METHOD SetPosition : BOOL
VAR_INPUT
	rPosition : LREAL;
END_VAR
// Start request once
IF NOT bSetPosRequested THEN
    bSetPosExecute   := TRUE;   // rising edge
    bSetPosRequested := TRUE;
END_IF

fbSetPos(Axis := Axis, Execute := bSetPosExecute, Position := rPosition, Mode := FALSE);

// Drop execute after it was accepted
IF fbSetPos.Busy THEN
    bSetPosExecute := FALSE;
END_IF

// Error handling
IF fbSetPos.Error THEN
    bSetPosExecute   := FALSE;
    bSetPosRequested := FALSE;   // ou mantenha TRUE se quiser retry controlado
    stStatus.eState  := E_ActuatorState.eError;
    stStatus.sMessage := 'Error in motor Set Position';
    SetPosition := FALSE;
    RETURN;
END_IF

// SUCCESS only on Done
IF fbSetPos.Done THEN
    bSetPosExecute   := FALSE;
    bSetPosRequested := FALSE;
    SetPosition := TRUE;
ELSE
    SetPosition := FALSE;
END_IF

(* Before Feb05th 2026
// Reuse the same logic from MoveAbsolute
IF NOT bSetPosRequested THEN
    bSetPosExecute := TRUE;
    bSetPosRequested := TRUE;
END_IF

// Call the internal motion block
fbSetPos(Axis := Axis, Execute := bSetPosExecute, Position := rPosition, Mode := FALSE);

// Update actuator status
stStatus.bBusy := fbSetPos.Busy;
stStatus.bDone := fbSetPos.Done;
stStatus.bError := fbSetPos.Error;
stStatus.iErrorCode := fbSetPos.ErrorID;

IF fbSetPos.busy THEN
    bSetPosExecute := FALSE;
END_IF

IF fbSetPos.Error THEN
    stStatus.eState := E_ActuatorState.eError;
    stStatus.sMessage := 'Error in motor Set Position';
END_IF

IF bSetPosRequested AND NOT fbSetPos.Busy AND NOT fbSetPos.Error THEN
    bSetPosRequested := FALSE;
    SetPosition := TRUE;
    RETURN;
ELSE
    SetPosition := FALSE;
END_IF
(*
// Call the internal motion block
fbSetPos(Axis := Axis, Execute := bSetPosExecute, Position := rPosition, Mode := FALSE);
*)*)
END_METHOD

METHOD Stop : BOOL
VAR_INPUT
END_VAR
VAR
END_VAR
// Default output value
Stop := FALSE;

// ============================================================================
// 1) First Stop trigger: set the request flag and generate the rising edge
//    on Execute for MC_Stop
// ============================================================================
IF NOT bStopRequested THEN
    bStopExecute  := TRUE;   // rising edge on MC_Stop.Execute
    bStopRequested := TRUE;
    bStopDone     := FALSE;
END_IF

// ============================================================================
// 2) Safety-net: if Stop was requested but the MC_Stop FB is idle,
//    without Done/Error, and Execute is FALSE (e.g., after a Reset),
//    then re-arm Execute to avoid getting stuck.
// ============================================================================
IF bStopRequested
   AND NOT fbStop.Busy
   AND NOT fbStop.Done
   AND NOT fbStop.Error
   AND NOT bStopExecute THEN
    bStopExecute := TRUE;
END_IF

// ============================================================================
// 3) Call the MC_Stop function block
// ============================================================================
fbStop(Axis := Axis, Execute := bStopExecute);

// ============================================================================
// 4) Internal Stop completion logic (Done / Requested)
// ============================================================================
IF fbStop.Done THEN
    bStopExecute := FALSE;      // release Execute after Done
    bStopDone    := TRUE;
END_IF

IF bStopDone AND NOT fbStop.Busy THEN
    bStopRequested := FALSE;    // stop procedure fully completed
END_IF

// ============================================================================
// 5) Error handling
// ============================================================================
stStatus.bError     := fbStop.Error;
stStatus.iErrorCode := fbStop.ErrorID;

IF fbStop.Error THEN
    stStatus.eState   := E_ActuatorState.eError;
    stStatus.sMessage := 'Error in Stop';
    // Stop remains FALSE; caller must handle Reset() afterwards
    RETURN;
END_IF

// ============================================================================
// 6) Successful completion: update status and return TRUE once
// ============================================================================
IF bStopDone AND NOT fbStop.Busy AND NOT bStopRequested THEN
    stStatus.bError     := FALSE;
    stStatus.iErrorCode := 0;
    stStatus.eState     := E_ActuatorState.eIdle;
    stStatus.sMessage   := 'Axis Stopped';

    // Prepare flags for the next Stop command
    bStopDone := FALSE;

    Stop := TRUE;   // Return TRUE for one cycle
    RETURN;
END_IF

// If execution reaches here, the Stop process is still ongoing
Stop := FALSE;


// Before - changed on Nov 20 2025
(* 
IF NOT bStopRequested THEN
	bStopExecute := TRUE;
	bStopRequested := TRUE;
END_IF

IF bStopRequested THEN
	fbStop(Axis := Axis, Execute := bStopExecute);
END_IF

IF bStopDone AND NOT fbStop.Busy THEN
	bStopRequested := FALSE;
END_IF

IF fbStop.Done THEN
	bStopExecute := FALSE;
	bStopDone := TRUE;
END_IF

stStatus.bError := fbStop.Error;
stStatus.iErrorCode := fbStop.ErrorID;

IF fbStop.Error THEN
	stStatus.eState := E_ActuatorState.eError;
	stStatus.sMessage := 'Error in Stop';
	Stop := FALSE;
END_IF

IF bStopDone AND NOT fbStop.Busy AND NOT bStopRequested THEN
	stStatus.bError := FALSE;
	stStatus.iErrorCode := 0;
	stStatus.eState := E_ActuatorState.eIdle;
	stStatus.sMessage := 'Axis Stopped';
	bStopDone := FALSE;
	Stop := TRUE;
	RETURN;
ELSE
	Stop := FALSE;
END_IF
*)
END_METHOD

END_FUNCTION_BLOCK

// ---- POUs/2. AutoCycle/Stages/FB_PostRun.TcPOU
FUNCTION_BLOCK FB_PostRun
VAR_INPUT
END_VAR
VAR_OUTPUT
END_VAR
VAR
END_VAR

END_FUNCTION_BLOCK

// ---- POUs/3. HMI/PRG_SetModulestatus.TcPOU
PROGRAM PRG_SetModulestatus
VAR
END_VAR

// Sets the Module status string based on the nTerminalState variable

// Terminal EK1100 EtherCAT Coupler
IF GVL_IO.nEK1100State = 8 THEN
	GVL_IO.sEK1100Status := 'Operational';
	ELSIF GVL_IO.nEK1100State = 4 THEN
 	GVL_IO.sEK1100Status := 'SAFEOP';
	ELSIF GVL_IO.nEK1100State = 3 THEN
 	GVL_IO.sEK1100Status := 'BOOT';
	ELSIF GVL_IO.nEK1100State = 2 THEN
 	GVL_IO.sEK1100Status := 'PREOP';
	ELSIF GVL_IO.nEK1100State = 1 THEN
 	GVL_IO.sEK1100Status := 'INIT';
END_IF

// TERMINAL - EL6070-0033	License Key Terminal for TwinCAT 3.1
IF GVL_IO.nEL6070State = 8 THEN
	GVL_IO.sEL6070Status := 'Operational';
	ELSIF GVL_IO.nEL6070State = 4 THEN
 	GVL_IO.sEL6070Status := 'SAFEOP';
	ELSIF GVL_IO.nEL6070State = 3 THEN
 	GVL_IO.sEL6070Status := 'BOOT';
	ELSIF GVL_IO.nEL6070State = 2 THEN
 	GVL_IO.sEL6070Status := 'PREOP';
	ELSIF GVL_IO.nEL6070State = 1 THEN
 	GVL_IO.sEL6070Status := 'INIT';
END_IF

// TERMINAL - EL6910 Safety PLC, 	Virtual Channels
IF GVL_IO.nEL6910State = 8 THEN
	GVL_IO.sEL6910Status := 'Operational';
	ELSIF GVL_IO.nEL6910State = 4 THEN
 	GVL_IO.sEL6910Status := 'SAFEOP';
	ELSIF GVL_IO.nEL6910State = 3 THEN
 	GVL_IO.sEL6910Status := 'BOOT';
	ELSIF GVL_IO.nEL6910State = 2 THEN
 	GVL_IO.sEL6910Status := 'PREOP';
	ELSIF GVL_IO.nEL6910State = 1 THEN
 	GVL_IO.sEL6910Status := 'INIT';
END_IF

// TERMINAL - EL1918_1 8-Channel Digital Safety Inputs
IF GVL_IO.nEL1918_1State = 8 THEN
	GVL_IO.sEL1918Status := 'Operational';
	ELSIF GVL_IO.nEL1918_1State = 4 THEN
 	GVL_IO.sEL1918Status := 'SAFEOP';
	ELSIF GVL_IO.nEL1918_1State = 3 THEN
 	GVL_IO.sEL1918Status := 'BOOT';
	ELSIF GVL_IO.nEL1918_1State = 2 THEN
 	GVL_IO.sEL1918Status := 'PREOP';
	ELSIF GVL_IO.nEL1918_1State = 1 THEN
 	GVL_IO.sEL1918Status := 'INIT';
END_IF

// TERMINAL - EL1918_2 8-Channel Digital Safety Inputs
IF GVL_IO.nEL1918_2State = 8 THEN
	GVL_IO.sEL1918_2Status := 'Operational';
	ELSIF GVL_IO.nEL1918_2State = 4 THEN
 	GVL_IO.sEL1918_2Status := 'SAFEOP';
	ELSIF GVL_IO.nEL1918_2State = 3 THEN
 	GVL_IO.sEL1918_2Status := 'BOOT';
	ELSIF GVL_IO.nEL1918_2State = 2 THEN
 	GVL_IO.sEL1918_2Status := 'PREOP';
	ELSIF GVL_IO.nEL1918_2State = 1 THEN
 	GVL_IO.sEL1918_2Status := 'INIT';
END_IF

// TERMINAL - EL2904 4-Channel Digital Output Terminal, TwinSAFE
IF GVL_IO.nEL2904State = 8 THEN
	GVL_IO.sEL2904Status := 'Operational';
	ELSIF GVL_IO.nEL2904State = 4 THEN
 	GVL_IO.sEL2904Status := 'SAFEOP';
	ELSIF GVL_IO.nEL2904State = 3 THEN
 	GVL_IO.sEL2904Status := 'BOOT';
	ELSIF GVL_IO.nEL2904State = 2 THEN
 	GVL_IO.sEL2904Status := 'PREOP';
	ELSIF GVL_IO.nEL2904State = 1 THEN
 	GVL_IO.sEL2904Status := 'INIT';
END_IF

// TERMINAL - EL2904_2 4-Channel Digital Output Terminal, TwinSAFE
IF GVL_IO.nEL2904_2State = 8 THEN
	GVL_IO.sEL2904_2Status := 'Operational';
	ELSIF GVL_IO.nEL2904_2State = 4 THEN
 	GVL_IO.sEL2904_2Status := 'SAFEOP';
	ELSIF GVL_IO.nEL2904_2State = 3 THEN
 	GVL_IO.sEL2904_2Status := 'BOOT';
	ELSIF GVL_IO.nEL2904_2State = 2 THEN
 	GVL_IO.sEL2904_2Status := 'PREOP';
	ELSIF GVL_IO.nEL2904_2State = 1 THEN
 	GVL_IO.sEL2904_2Status := 'INIT';
END_IF

// TERMINAL - EL1809_1 16-Channel Digital Input Terminal
IF GVL_IO.nEL1809State = 8 THEN
	GVL_IO.sEL1809Status := 'Operational';
	ELSIF GVL_IO.nEL1809State = 4 THEN
 	GVL_IO.sEL1809Status := 'SAFEOP';
	ELSIF GVL_IO.nEL1809State = 3 THEN
 	GVL_IO.sEL1809Status := 'BOOT';
	ELSIF GVL_IO.nEL1809State = 2 THEN
 	GVL_IO.sEL1809Status := 'PREOP';
	ELSIF GVL_IO.nEL1809State = 1 THEN
 	GVL_IO.sEL1809Status := 'INIT';
END_IF

// TERMINAL - EL2809_1	16-Channel Digital Output Terminal
IF GVL_IO.nEL2809State = 8 THEN
	GVL_IO.sEL2809Status := 'Operational';
	ELSIF GVL_IO.nEL2809State = 4 THEN
 	GVL_IO.sEL2809Status := 'SAFEOP';
	ELSIF GVL_IO.nEL2809State = 3 THEN
 	GVL_IO.sEL2809Status := 'BOOT';
	ELSIF GVL_IO.nEL2809State = 2 THEN
 	GVL_IO.sEL2809Status := 'PREOP';
	ELSIF GVL_IO.nEL2809State = 1 THEN
 	GVL_IO.sEL2809Status := 'INIT';
END_IF

// TERMINAL - EL3058	8-Channel Analog Input Terminal 4…20mA 12 Bit
IF GVL_IO.nEL3058State = 8 THEN
	GVL_IO.sEL3058Status := 'Operational';
	ELSIF GVL_IO.nEL3058State = 4 THEN
 	GVL_IO.sEL3058Status := 'SAFEOP';
	ELSIF GVL_IO.nEL3058State = 3 THEN
 	GVL_IO.sEL3058Status := 'BOOT';
	ELSIF GVL_IO.nEL3058State = 2 THEN
 	GVL_IO.sEL3058Status := 'PREOP';
	ELSIF GVL_IO.nEL3058State = 1 THEN
 	GVL_IO.sEL3058Status := 'INIT';
END_IF

// Terminal EL3058 8-Channel Analog Input Terminal 4…20mA 12 Bit (Term 10)
IF GVL_IO.nEL3058State = 8 THEN
	GVL_IO.sEL3058Status := 'Operational';
	ELSIF GVL_IO.nEL3058State = 4 THEN
 	GVL_IO.sEL3058Status := 'SAFEOP';
	ELSIF GVL_IO.nEL3058State = 3 THEN
 	GVL_IO.sEL3058Status := 'BOOT';
	ELSIF GVL_IO.nEL3058State = 2 THEN
 	GVL_IO.sEL3058Status := 'PREOP';
	ELSIF GVL_IO.nEL3058State = 1 THEN
 	GVL_IO.sEL3058Status := 'INIT';
END_IF

// Terminal EL6002	2-channel Serial Interface RS232, D-sub Connection (Term 11)
IF GVL_IO.nEL6002State = 8 THEN
	GVL_IO.sEL6002Status := 'Operational';
	ELSIF GVL_IO.nEL6002State = 4 THEN
 	GVL_IO.sEL6002Status := 'SAFEOP';
	ELSIF GVL_IO.nEL6002State = 3 THEN
 	GVL_IO.sEL6002Status := 'BOOT';
	ELSIF GVL_IO.nEL6002State = 2 THEN
 	GVL_IO.sEL6002Status := 'PREOP';
	ELSIF GVL_IO.nEL6002State = 1 THEN
 	GVL_IO.sEL6002Status := 'INIT';
END_IF

END_PROGRAM

// ---- POUs/7. EventsAndAlarms/FB_AlarmHandler.TcPOU
FUNCTION_BLOCK FB_AlarmHandler EXTENDS FB_TcAlarm
VAR_INPUT
	evtEntry	: TcEventEntry;
	bEvt		: BOOL;
	bConfirm	: BOOL;
	sSystem		: STRING; // Adding Alarm system name
	sMessage	: STRING; // Alarm Message
END_VAR
VAR_OUTPUT
END_VAR
VAR
	bInit	: BOOL := TRUE;
	bMem	: BOOL;
END_VAR

IF bInit THEN
	SUPER^.CreateEx(evtEntry, TRUE, 0);
	bInit	:= FALSE;
END_IF

// To when the alarm is triggered for the first time
IF bEvt AND NOT bMem AND SUPER^.eConfirmationState <> TcEventConfirmationState.WaitForConfirmation THEN
	SUPER^.ipArguments.AddString(sSystem).AddString(sMessage); // Adiciona as strings ao alarme
	SUPER^.Raise(0);
END_IF

// To when the alarm is reset
IF bMem AND NOT bEvt THEN
	SUPER^.Clear(0, FALSE);
END_IF

// Alarm confirmation
IF bConfirm THEN
	SUPER^.Confirm(0);
END_IF

bMem := bEvt;

END_FUNCTION_BLOCK

// ---- POUs/7. EventsAndAlarms/FB_ErrorHandler.TcPOU
FUNCTION_BLOCK FB_ErrorHandler

VAR_INPUT
END_VAR

VAR_OUTPUT
	bErrorResolved : BOOL;
END_VAR

VAR
END_VAR

//bErrorResolved := (* Verdadeiro quando o erro for resolvido

END_FUNCTION_BLOCK

// ---- POUs/Functions/F_REAL_TO_STRING_2DEC.TcPOU
FUNCTION F_REAL_TO_STRING_2DEC : STRING
VAR_INPUT
	rInput : REAL;
END_VAR
VAR
	iInt    : DINT;
    iDec    : DINT;
    rTmp    : REAL;
END_VAR

iInt := TRUNC(rInput);
rTmp := ABS(rInput - iInt);            // decimal part
iDec := TRUNC((rTmp * 100.0) + 0.5);   // manual rounding

IF rInput >= 0.0 THEN
    F_REAL_TO_STRING_2DEC := CONCAT( DINT_TO_STRING(iInt), CONCAT('.', DINT_TO_STRING(iDec)) );
ELSE
    F_REAL_TO_STRING_2DEC := CONCAT('-', CONCAT( DINT_TO_STRING(ABS(iInt)), CONCAT('.', DINT_TO_STRING(iDec)) ));
END_IF

END_FUNCTION

// ---- POUs/Functions/F_SqlEscapeString.TcPOU
FUNCTION F_SqlEscapeString : STRING
VAR_INPUT
	sInput : STRING(500);
END_VAR
VAR
	i       : INT;
    sChar   : STRING(1);
    sOutput : STRING(500);
END_VAR

sOutput := '';

FOR i := 1 TO LEN(sInput) DO
    sChar := MID(sInput, 1, i);

    IF sChar = '$'' THEN
        sOutput := CONCAT(sOutput, '$'$'');
    ELSE
        sOutput := CONCAT(sOutput, sChar);
    END_IF
END_FOR

F_SqlEscapeString := sOutput;

END_FUNCTION

// ---- POUs/Levels/FB_LevelSensors.TcPOU
FUNCTION_BLOCK FB_LevelSensors
VAR_INPUT
	abyInputs : ARRAY[1..5, 0..3] OF BYTE; // 5 sensors, 4 bytes each
    eSensorID : E_LevelSensorID;
END_VAR
VAR_OUTPUT
	stLevelData : ST_KQ1000_Data;
END_VAR
VAR
	fbParsers : ARRAY[1..5] OF FB_KQ1000_Parser;
    i : INT;
END_VAR

// Parsers execute
FOR i := 1 TO 5 DO
    fbParsers[i].byInput0 := abyInputs[i, 0];
    fbParsers[i].byInput1 := abyInputs[i, 1];
    fbParsers[i].byInput2 := abyInputs[i, 2];
    fbParsers[i].byInput3 := abyInputs[i, 3];
END_FOR

// Sends the result based on sensor id
stLevelData := fbParsers[eSensorID].stData;

END_FUNCTION_BLOCK

// ---- POUs/MARCO/OLD/POU_Master_Calib.TcPOU
PROGRAM POU_Master_Calib
VAR
	criteria: REAL := 0.5; // Acceptance Criteria (0.1 ~ 5.0)
	failures: INT := 0; // Allowable Failures (0 ~ 5)
	targetVolume: REAL := 0.50; // Volume Target (mL)
	replicates: INT := 2; // Number of checks (0 ~ 10)
	tareWt: REAL; //Weight before
	grossWt: REAL; //Weight after
	netWt: REAL; // rsult of (grossWt - tareWt)
	netVolume: REAL; //result of (netWt * density)
	state: INT;
	valveNo: INT;
	pumpNo: INT:=1;
	timeWt: ton;
	timer2: ton;
	timer3: ton;
	selectPump: ARRAY[1..10] OF STRING;
	result: ARRAY[1..10] OF ST_Results;
	start: BOOL;
	stop: BOOL;
	movimentDONE: BOOL;
	revs: REAL;
	valvePos: USINT;
	repli: INT:= 1;
	axiPower: MC_Power;
	i: INT;
	scale: FB_ScaleDevice;
	adjust: ARRAY[1..10] OF BOOL;
	correctRev: REAL;
	enableAdj: BOOL;
	opening: REAL;
	runLinear: BOOL;
	adjustSum: REAL;
	recResult: int:=1;
END_VAR

timeWt();
timer2();
timer3();

IF stop THEN
	powerOFF();
	stop:=FALSE;
END_IF

IF pumpNo = 1 OR pumpNo = 2 THEN
	valveNo:= 1;
ELSIF pumpNo = 3 OR pumpNo = 4 THEN
	valveNo:= 2;
ELSIF pumpNo = 5 OR pumpNo = 6 THEN
	valveNo:= 3;
ELSIF pumpNo = 7 OR pumpNo = 8 THEN
	valveNo:= 4;
ELSIF pumpNo = 9 OR pumpNo = 10 THEN
	valveNo:= 5;
END_IF

CASE state OF
	
0: //Idle
	IF start THEN
		GVL_Marco.revs:= GVL_Marco.mL_target;
		GVL_Marco.valvPos:= 6;
		timeWt(in:=TRUE, pt:=T#10S);
		repli:= 1;
		recResult:= 1;
		
		FOR i:= 1 TO 10 BY 1 DO
			GVL_Marco.resetAxi[i]:= FALSE;
			GVL_Marco.enableAxi[i]:= TRUE;
		END_FOR 
		
		FOR i:= 1 TO 5 BY 1 DO
			GVL_Marco.enableValv[i]:= TRUE;		
		END_FOR
		
		FOR i:=1 TO 50 BY 1 DO
			GVL_Marco.calibResult[i].grossWt:=0;
			GVL_Marco.calibResult[i].netWt:=0;
			GVL_Marco.calibResult[i].pumpNo:=0;
			GVL_Marco.calibResult[i].tareWt:=0;
		END_FOR
		
		state:= 10;
	ELSE
		state:= 0;
	END_IF
	
10:	//Disable valves
	
	IF GVL_Motion.aValves[1].Axis.Status.InTargetPosition AND
		GVL_Motion.aValves[2].Axis.Status.InTargetPosition AND
		GVL_Motion.aValves[3].Axis.Status.InTargetPosition AND
		GVL_Motion.aValves[4].Axis.Status.InTargetPosition AND
		GVL_Motion.aValves[5].Axis.Status.InTargetPosition AND timeWt.Q THEN
		FOR i:= 1 TO 5 BY 1 DO
			GVL_Marco.enableValv[i]:= FALSE;		
		END_FOR
		timeWt(in:=FALSE);
		timer3(in:=TRUE, pt:=T#10S);
		state:= 20;
	ELSE
		state:= 10;
	END_IF		

20:	//Fill Jar from Box
	
	IF NOT GVL_Motion.aPumps[pumpNo].Rotary.Axis.Status.Disabled AND (timer3.Q OR timeWt.Q) THEN
		IF repli < 2 THEN
		revs:= GVL_Marco.revs*2.4;	
		END_IF
		GVL_Marco.runFWD[pumpNo]:= TRUE;
		timer3(in:=FALSE);
		start:= FALSE;
		timer2(in:=TRUE, pt:=T#10S);
		state:= 30;
	ELSE
		state:= 20;
	END_IF

30: //Waiting

	IF GVL_Motion.aPumps[pumpNo].Rotary.Axis.Status.NotMoving AND timer2.Q THEN
		GVL_Marco.runFWD[pumpNo]:= FALSE;
		timer2(in:=FALSE);
		timeWt(in:=TRUE, pt:=T#10S);
		GVL_Calibration.fbScaleDevice.RequestWeight();
		state:= 40;
	ELSE
		state:= 30;
	END_IF
	
40: //Make Tara
	
	IF timeWt.Q THEN
		tareWt:= GVL_Calibration.fbScaleDevice.RequestWeight();
		timeWt(in:=FALSE);
		state:= 50;
	ELSE
		state:= 40;
	END_IF
	
50: //Fill box from jar

	IF tareWt <> 9999.0 THEN
		GVL_Marco.calibResult[recResult].tareWt:= tareWt;
		revs:= GVL_Marco.revs;
		GVL_Marco.runBWD[pumpNo]:= TRUE;
		timer2(in:=TRUE, pt:=T#10S);
		state:= 60;
	ELSE
		state:= 50;
	END_IF
	
60: //Waiting

	IF NOT GVL_Motion.aPumps[pumpNo].Rotary.Axis.Status.Moving AND timer2.Q THEN
		GVL_Marco.runBWD[pumpNo]:= FALSE;
		timer2(in:=FALSE);
		timeWt(in:=TRUE, pt:=T#10S);
		GVL_Calibration.fbScaleDevice.RequestWeight();
		state:= 70;
	ELSE
		state:= 60;
	END_IF

70: //Get gross weight
	
	IF timeWt.Q THEN
		grossWt:= GVL_Calibration.fbScaleDevice.RequestWeight();
		timeWt(in:=FALSE);
		state:= 80;
	ELSE
		state:= 70;
	END_IF
	
80: //Return jar to box

	IF grossWt <> 9999.0 THEN
		GVL_Marco.calibResult[recResult].grossWt:= grossWt;
		GVL_Marco.calibResult[recResult].netWt:= GVL_Marco.calibResult[recResult].grossWt - GVL_Marco.calibResult[recResult].tareWt;
		GVL_Marco.calibResult[recResult].pumpNo:= pumpNo;
		recResult:= recResult +1;
			
		//revs:= GVL_Marco.revs;
		//GVL_Marco.runFWD[pumpNo]:= TRUE;

		timer3(in:=TRUE, pt:=T#10S);
		repli := repli +1; 
		state:= 90;
	ELSE
		state:= 80;
	END_IF

90: //Check replicates

	IF repli < replicates+1 AND timer3.Q AND GVL_Motion.aPumps[pumpNo].Rotary.Axis.Status.NotMoving THEN //Return to the next replicate
		timer3(in:=FALSE);
		timeWt(in:=TRUE, pt:=T#10S);
		GVL_Marco.runFWD[pumpNo]:= FALSE;
		state:= 20;
	ELSIF repli >= replicates AND timer3.Q AND GVL_Motion.aPumps[pumpNo].Rotary.Axis.Status.NotMoving THEN //Empty the jar to box
		timer3(in:=FALSE);
		GVL_Marco.runFWD[pumpNo]:= FALSE;
		revs:= GVL_Marco.revs*2.4;
		GVL_Marco.runBWD[pumpNo]:= TRUE;
		timer2(in:=TRUE, pt:=T#10S);
		state:= 100;
	ELSE
		state:= 90;
	END_IF

100: 

	IF  GVL_Motion.aPumps[pumpNo].Rotary.Axis.Status.NotMoving AND timer2.Q THEN
		timer2(in:=FALSE);
		IF pumpNo = 10 THEN
			GVL_Marco.runBWD[pumpNo]:= FALSE;
			timer3(in:=TRUE, pt:=T#10S);
			state:= 110;
		ELSE
			pumpNo:= pumpNo + 1;
			repli:= 1;
			timer3(in:=TRUE, pt:=T#10S);
			state:= 20;
		END_IF
		
	ELSE
		state:= 100;
	END_IF
	
110: //Done

	IF GVL_Motion.aPumps[1].Rotary.Axis.Status.NotMoving AND
		GVL_Motion.aPumps[2].Rotary.Axis.Status.NotMoving AND
		GVL_Motion.aPumps[3].Rotary.Axis.Status.NotMoving AND
		GVL_Motion.aPumps[4].Rotary.Axis.Status.NotMoving AND
		GVL_Motion.aPumps[5].Rotary.Axis.Status.NotMoving AND
		GVL_Motion.aPumps[6].Rotary.Axis.Status.NotMoving AND
		GVL_Motion.aPumps[7].Rotary.Axis.Status.NotMoving AND
		GVL_Motion.aPumps[8].Rotary.Axis.Status.NotMoving AND
		GVL_Motion.aPumps[9].Rotary.Axis.Status.NotMoving AND
		GVL_Motion.aPumps[10].Rotary.Axis.Status.NotMoving AND timer3.Q THEN
		FOR i:=1 TO 10 BY 1 DO
			GVL_Marco.runBWD[i]:= FALSE;
		END_FOR
		
		timer3(in:=FALSE);
		timeWt(in:=TRUE, pt:=T#10S);
		state:= 120;
	ELSE
		state:= 110;
	END_IF
	
120:

	IF GVL_Motion.aPumps[1].Rotary.Axis.Status.NotMoving AND
		GVL_Motion.aPumps[2].Rotary.Axis.Status.NotMoving AND
		GVL_Motion.aPumps[3].Rotary.Axis.Status.NotMoving AND
		GVL_Motion.aPumps[4].Rotary.Axis.Status.NotMoving AND
		GVL_Motion.aPumps[5].Rotary.Axis.Status.NotMoving AND
		GVL_Motion.aPumps[6].Rotary.Axis.Status.NotMoving AND
		GVL_Motion.aPumps[7].Rotary.Axis.Status.NotMoving AND
		GVL_Motion.aPumps[8].Rotary.Axis.Status.NotMoving AND
		GVL_Motion.aPumps[9].Rotary.Axis.Status.NotMoving AND
		GVL_Motion.aPumps[10].Rotary.Axis.Status.NotMoving AND timeWt.Q THEN
		FOR i:=1 TO 10 BY 1 DO
			GVL_Marco.resetAxi[i]:= TRUE;
			GVL_Marco.enableAxi[i]:= FALSE;
		END_FOR
		
		(*IF GVL_Marco.revs > GVL_Marco.mL_target THEN
			correctRev:= GVL_Marco.revs - GVL_Marco.mL_target;
		ELSIF GVL_Marco.revs < GVL_Marco.mL_target THEN
			correctRev:= GVL_Marco.mL_target - GVL_Marco.revs; 	
		END_IF*)
		state:= 0;
	ELSE
		state:= 120;
	END_IF
	
END_CASE

METHOD moveValve : BOOL
VAR
	state: INT;
	valveNo: INT;
END_VAR
VAR_INPUT
	pumNo: INT;
	valvePos: USINT;
	
END_VAR
IF pumpNo = 1 OR pumpNo = 2 THEN
	valveNo:= 1;
ELSIF pumpNo = 3 OR pumpNo = 4 THEN
	valveNo:= 2;
ELSIF pumpNo = 5 OR pumpNo = 6 THEN
	valveNo:= 3;
ELSIF pumpNo = 7 OR pumpNo = 8 THEN
	valveNo:= 4;
ELSIF pumpNo = 9 OR pumpNo = 10 THEN
	valveNo:= 5;
END_IF

GVL_Motion.aValvesObj[valveNo].MoveValve(iPosition := valvePos, rVelocity := GVL_Motion.aValves[1].rTargetVel, rAcc := GVL_Motion.aValves[1].rAcceleration, rDec := GVL_Motion.aValves[1].rDeceleration);

CASE state OF
	
0:

	IF NOT GVL_Motion.aValves[valveNo].Axis.Status.Moving THEN
		GVL_Motion.aValvesObj[valveNo].MoveValve(iPosition := valvePos, rVelocity := GVL_Motion.aValves[1].rTargetVel, rAcc := GVL_Motion.aValves[1].rAcceleration, rDec := GVL_Motion.aValves[1].rDeceleration);
		movimentDONE:=FALSE;
		state:= 1;
	ELSE
		state:= 0;	
	END_IF

1:
	IF NOT GVL_Motion.aValves[valveNo].Axis.Status.Moving THEN
			movimentDONE:= TRUE;
			State:= 0;
		ELSE
			state:= 1;
		END_IF
	
	
END_CASE
END_METHOD

METHOD powerOFF : BOOL
VAR
	axiPower: MC_Power;
	pumpNo: INT;
	
END_VAR
VAR_INPUT
	
	
END_VAR
FOR pumpNo:=1 TO 10 BY 1 DO
	axiPower(
	Axis:= GVL_Motion.aPumps[pumpNo].Rotary.Axis,
	Enable:= FALSE,
	Enable_Negative:= FALSE,
	Enable_Positive:= FALSE,
	Override:= 100);
	
	axiPower(
	Axis:= GVL_Motion.aPumps[pumpNo].Linear.Axis,
	Enable:= FALSE,
	Enable_Negative:= FALSE,
	Enable_Positive:= FALSE,
	Override:= 100);
END_FOR
END_METHOD

METHOD runBwd : BOOL
VAR
	moveRel: MC_MoveRelative;
	selectPosRel: LREAL;
	
END_VAR
VAR_INPUT
	pumpNo: INT;
	revs: INT;
	 
END_VAR

selectPosRel:= revs*360;

moveRel(
	Axis:= GVL_Motion.aPumps[pumpNo].Rotary.Axis,
	Execute:= TRUE,
	Distance:= selectPosRel*-1,
	Velocity:= 3000,
	Acceleration:= 3000,
	Deceleration:= 3000);
END_METHOD

METHOD runFwd : BOOL
VAR
	moveRel: MC_MoveRelative;
	selectPosRel: LREAL;
	
END_VAR
VAR_INPUT
	pumpNo: INT;
	revs: INT;
	 
END_VAR

selectPosRel:= revs*360;

moveRel(
	Axis:= GVL_Motion.aPumps[pumpNo].Rotary.Axis,
	Execute:= TRUE,
	Distance:= selectPosRel,
	Velocity:= 3000,
	Acceleration:= 3000,
	Deceleration:= 3000);
END_METHOD

END_PROGRAM

// ---- POUs/MARCO/OLD/POU_Master_Calib_1.TcPOU
PROGRAM POU_Master_Calib_1
VAR
	criteria: REAL := 0.5; // Acceptance Criteria (0.1 ~ 5.0)
	failures: INT := 0; // Allowable Failures (0 ~ 5)
	targetVolume: REAL := 0.50; // Volume Target (mL)
	replicates: INT := 5; // Number of checks (0 ~ 10)
	tareWt: REAL; //Weight before
	grossWt: REAL; //Weight after
	netWt: REAL; // rsult of (grossWt - tareWt)
	netVolume: REAL; //result of (netWt * density)
	state: INT;
	valveNo: INT;
	pumpNo: INT:=1;
	timeWt: ton;
	timer2: ton;
	timer3: ton;
	selectPump: ARRAY[1..10] OF STRING;
	result: ARRAY[1..50] OF ST_Results;
	start: BOOL;
	stop: BOOL;
	movimentDONE: BOOL;
	revs: REAL;
	valvePos: USINT;
	repli: INT:= 1;
	axiPower: MC_Power;
	i: INT;
	scale: FB_ScaleDevice;
	adjust: ARRAY[1..10] OF BOOL;
	correctRev: REAL;
	enableAdj: BOOL;
	opening: REAL;
	runLinear: BOOL;
	adjustSum: REAL;
END_VAR

timeWt();
timer2();
timer3();

IF stop THEN
	powerOFF();
	stop:=FALSE;
END_IF

IF pumpNo = 1 OR pumpNo = 2 THEN
	valveNo:= 1;
ELSIF pumpNo = 3 OR pumpNo = 4 THEN
	valveNo:= 2;
ELSIF pumpNo = 5 OR pumpNo = 6 THEN
	valveNo:= 3;
ELSIF pumpNo = 7 OR pumpNo = 8 THEN
	valveNo:= 4;
ELSIF pumpNo = 9 OR pumpNo = 10 THEN
	valveNo:= 5;
END_IF

CASE state OF
	
0: //Idle
	IF start THEN
		GVL_Marco.revs:= GVL_Marco.mL_target;
		GVL_Marco.resetAxi:= FALSE;
		GVL_Marco.valvPos:= 2;
		GVL_Marco.enableValv:= TRUE;
		timeWt(in:=TRUE, pt:=T#10S);
		GVL_Marco.enableAxi:= TRUE;
		FOR i:=1 TO 10 BY 1 DO
			result[i].gross:= 0;
			result[i].rest:= 0;
			result[i].tare:= 0;
		END_FOR
		repli:= 1;
		state:= 10;
	ELSE
		state:= 0;
	END_IF
	
10:	//Enable the pump motor
	
	IF GVL_Motion.aValves[valveNo].Axis.Status.InTargetPosition AND timeWt.Q THEN
		GVL_Marco.enableValv:= FALSE;
		timeWt(in:=FALSE);
		IF pumpNo >= 10 THEN
			pumpNo:= 2;
			state:= 20;
		ELSE
			pumpNo:= pumpNo + 1;
			state:= 0;
		END_IF
	ELSE
		state:= 10;
	END_IF		

20:	//Fill the Jars from Bottle
	
	IF NOT GVL_Motion.aPumps[pumpNo].Rotary.Axis.Status.Disabled AND timer2.Q THEN
		revs:= GVL_Marco.revs*2.4;
		GVL_Marco.runFWD:= TRUE;
		timer2(in:=TRUE, pt:=T#10S);
		IF pumpNo >= 10 THEN
			pumpNo:= 2;
			start:= FALSE;
			state:= 30;
		ELSE
			timer2(in:=FALSE);
			pumpNo:= pumpNo + 1;
			GVL_Marco.runFWD:= FALSE;
			state:= 20;
		END_IF
	ELSE
		state:= 20;
	END_IF

30: //Move valve to position 6
	
	IF NOT GVL_Motion.aPumps[pumpNo].Rotary.Axis.Status.Moving AND timer2.Q THEN
		GVL_Marco.runFWD:= FALSE;
		GVL_Marco.valvPos:= 6;
		GVL_Marco.enableValv:= TRUE;
		timer2(in:=FALSE);
		timeWt(in:=TRUE, pt:=T#10S);
		IF pumpNo >= 10 THEN
			pumpNo:= 2;
			state:= 40;
		ELSE
			pumpNo:= pumpNo + 1;
			state:= 30;
		END_IF
	ELSE
		state:= 30;
	END_IF


40: //Fill the calibration box( SETUP )

	IF GVL_Motion.aValves[valveNo].Axis.Status.InTargetPosition AND timeWt.Q THEN
		GVL_Marco.enableValv:= FALSE;
		revs:= GVL_Marco.revs/2;
		GVL_Marco.runBWD:= TRUE;
		timeWt(in:=FALSE);
		timer2(in:=TRUE, pt:=T#5S);
		state:= 50;
		
	ELSE
		state:= 40;	
	END_IF

50: //Waiting

	IF NOT GVL_Motion.aPumps[pumpNo].Rotary.Axis.Status.Moving AND timer2.Q THEN
		GVL_Marco.runBWD:= FALSE;
		timer2(in:=FALSE);
		timeWt(in:=TRUE, pt:=T#10S);
		GVL_Calibration.fbScaleDevice.RequestWeight();
		state:= 55;
	ELSE
		state:= 50;
	END_IF
	
55: //Make Tara
	
	IF timeWt.Q THEN
		tareWt:= GVL_Calibration.fbScaleDevice.RequestWeight();
		timeWt(in:=FALSE);
		state:= 60;
	ELSE
		state:= 55;
	END_IF
	
60: //Fill calibration box

	IF tareWt <> 9999.0 THEN
		result[repli].tare:= tareWt;
		revs:= GVL_Marco.revs;
		GVL_Marco.runBWD:= TRUE;
		timer2(in:=TRUE, pt:=T#5S);
		state:= 70;
	ELSE
		state:= 60;
	END_IF
	
70: //Waiting

	IF NOT GVL_Motion.aPumps[pumpNo].Rotary.Axis.Status.Moving AND timer2.Q THEN
		GVL_Marco.runBWD:= FALSE;
		timer2(in:=FALSE);
		timeWt(in:=TRUE, pt:=T#10S);
		GVL_Calibration.fbScaleDevice.RequestWeight();
		state:= 75;
	ELSE
		state:= 70;
	END_IF

75: //Get gross weight
	
	IF timeWt.Q THEN
		grossWt:= GVL_Calibration.fbScaleDevice.RequestWeight();
		timeWt(in:=FALSE);
		state:= 80;
	ELSE
		state:= 75;
	END_IF
	
80: //Return solvent to jar

	IF grossWt <> 9999.0 THEN
		result[repli].gross:= grossWt;
		result[repli].rest:= result[repli].gross - result[repli].tare;
		netWt:= result[repli].rest;
			IF (netWt > GVL_Marco.mL_target+((GVL_Marco.mL_target*0.5)/100) OR netWt < GVL_Marco.mL_target-((GVL_Marco.mL_target*0.5)/100)) THEN
				adjust[repli]:= TRUE;
			ELSE
				adjust[repli]:= FALSE;
			END_IF
			IF repli >= replicates THEN
				revs:= GVL_Marco.revs*2;
				GVL_Marco.runFWD:= TRUE;
			ELSE
				revs:= GVL_Marco.revs;
				GVL_Marco.runFWD:= TRUE;
			END_IF
		timer3(in:=TRUE, pt:=T#10S);
		repli := repli +1;
		state:= 90;
	ELSE
		state:= 80;
	END_IF

90: //Check replicates

	IF repli < replicates+1 AND timer3.Q AND GVL_Motion.aPumps[pumpNo].Rotary.Axis.Status.NotMoving THEN
		timer3(in:=FALSE);
		GVL_Marco.runFWD:= FALSE;
		timer2(in:=TRUE, pt:=T#5S);
		state:= 50;
	ELSIF repli >= replicates AND timer3.Q AND GVL_Motion.aPumps[pumpNo].Rotary.Axis.Status.NotMoving THEN
		timer3(in:=FALSE);
		GVL_Marco.runFWD:= FALSE;
		GVL_Marco.valvPos:= 2;
		GVL_Marco.enableValv:= TRUE;
		timer2(in:=TRUE, pt:=T#10S);
		IF pumpNo >= 10 THEN
			pumpNo:= 2;
			state:= 100;
		ELSE
			pumpNo:= pumpNo + 1;
			repli:= 1;
			state:= 50;
		END_IF
	ELSE
		state:= 90;
	END_IF

100: //Empty the jar

	IF  GVL_Motion.aValves[valveNo].Axis.Status.InTargetPosition AND timer2.Q THEN
		GVL_Marco.enableValv:= FALSE;
		revs:= GVL_Marco.revs*2.4;
		GVL_Marco.runBWD:= TRUE;
		timer2(in:=FALSE);
		timer3(in:=TRUE, pt:=T#10S);
		IF pumpNo >= 10 THEN
			pumpNo:= 2;
			state:= 110;
		ELSE
			pumpNo:= pumpNo + 1;
			state:= 100;
		END_IF
	ELSE
		state:= 100;
	END_IF
	
110: //Done

	IF NOT GVL_Motion.aPumps[pumpNo].Rotary.Axis.Status.Moving AND timer3.Q THEN
		GVL_Marco.runBWD:= FALSE;
		timer3(in:=FALSE);
		timeWt(in:=TRUE, pt:=T#10S);
		IF pumpNo >= 10 THEN
			pumpNo:= 2;
			state:= 120;
		ELSE
			pumpNo:= pumpNo + 1;
			state:= 110;
		END_IF
	ELSE
		state:= 110;
	END_IF
	
120:

	IF GVL_Motion.aPumps[pumpNo].Rotary.Axis.Status.NotMoving AND timeWt.Q THEN
		GVL_Marco.resetAxi:= TRUE;
		GVL_Marco.enableAxi:= FALSE;
		IF pumpNo >= 10 THEN
			pumpNo:= 2;
			state:= 0;
		ELSE
			pumpNo:= pumpNo + 1;
			state:= 120;
		END_IF
	ELSE
		state:= 120;
	END_IF
	
END_CASE

METHOD moveValve : BOOL
VAR
	state: INT;
	valveNo: INT;
END_VAR
VAR_INPUT
	pumNo: INT;
	valvePos: USINT;
	
END_VAR
IF pumpNo = 1 OR pumpNo = 2 THEN
	valveNo:= 1;
ELSIF pumpNo = 3 OR pumpNo = 4 THEN
	valveNo:= 2;
ELSIF pumpNo = 5 OR pumpNo = 6 THEN
	valveNo:= 3;
ELSIF pumpNo = 7 OR pumpNo = 8 THEN
	valveNo:= 4;
ELSIF pumpNo = 9 OR pumpNo = 10 THEN
	valveNo:= 5;
END_IF

GVL_Motion.aValvesObj[valveNo].MoveValve(iPosition := valvePos, rVelocity := GVL_Motion.aValves[1].rTargetVel, rAcc := GVL_Motion.aValves[1].rAcceleration, rDec := GVL_Motion.aValves[1].rDeceleration);

CASE state OF
	
0:

	IF NOT GVL_Motion.aValves[valveNo].Axis.Status.Moving THEN
		GVL_Motion.aValvesObj[valveNo].MoveValve(iPosition := valvePos, rVelocity := GVL_Motion.aValves[1].rTargetVel, rAcc := GVL_Motion.aValves[1].rAcceleration, rDec := GVL_Motion.aValves[1].rDeceleration);
		movimentDONE:=FALSE;
		state:= 1;
	ELSE
		state:= 0;	
	END_IF

1:
	IF NOT GVL_Motion.aValves[valveNo].Axis.Status.Moving THEN
			movimentDONE:= TRUE;
			State:= 0;
		ELSE
			state:= 1;
		END_IF
	
	
END_CASE
END_METHOD

METHOD powerOFF : BOOL
VAR
	axiPower: MC_Power;
	pumpNo: INT;
	
END_VAR
VAR_INPUT
	
	
END_VAR
FOR pumpNo:=1 TO 10 BY 1 DO
	axiPower(
	Axis:= GVL_Motion.aPumps[pumpNo].Rotary.Axis,
	Enable:= FALSE,
	Enable_Negative:= FALSE,
	Enable_Positive:= FALSE,
	Override:= 100);
	
	axiPower(
	Axis:= GVL_Motion.aPumps[pumpNo].Linear.Axis,
	Enable:= FALSE,
	Enable_Negative:= FALSE,
	Enable_Positive:= FALSE,
	Override:= 100);
END_FOR
END_METHOD

METHOD runBwd : BOOL
VAR
	moveRel: MC_MoveRelative;
	selectPosRel: LREAL;
	
END_VAR
VAR_INPUT
	pumpNo: INT;
	revs: INT;
	 
END_VAR

selectPosRel:= revs*360;

moveRel(
	Axis:= GVL_Motion.aPumps[pumpNo].Rotary.Axis,
	Execute:= TRUE,
	Distance:= selectPosRel*-1,
	Velocity:= 3000,
	Acceleration:= 3000,
	Deceleration:= 3000);
END_METHOD

METHOD runFwd : BOOL
VAR
	moveRel: MC_MoveRelative;
	selectPosRel: LREAL;
	
END_VAR
VAR_INPUT
	pumpNo: INT;
	revs: INT;
	 
END_VAR

selectPosRel:= revs*360;

moveRel(
	Axis:= GVL_Motion.aPumps[pumpNo].Rotary.Axis,
	Execute:= TRUE,
	Distance:= selectPosRel,
	Velocity:= 3000,
	Acceleration:= 3000,
	Deceleration:= 3000);
END_METHOD

END_PROGRAM

// ---- POUs/MARCO/OLD/POU_Master_Calib_2.TcPOU
PROGRAM POU_Master_Calib_2
VAR
	criteria: REAL := 0.5; // Acceptance Criteria (0.1 ~ 5.0)
	failures: INT := 0; // Allowable Failures (0 ~ 5)
	targetVolume: REAL := 0.50; // Volume Target (mL)
	replicates: INT := 5; // Number of checks (0 ~ 10)
	tareWt: REAL; //Weight before
	grossWt: REAL; //Weight after
	netWt: REAL; // rsult of (grossWt - tareWt)
	netVolume: REAL; //result of (netWt * density)
	state: INT;
	valveNo: INT;
	pumpNo: INT:=1;
	timeWt: ton;
	timer2: ton;
	timer3: ton;
	selectPump: ARRAY[1..10] OF STRING;
	result: ARRAY[1..10] OF ST_Results;
	start: BOOL;
	stop: BOOL;
	movimentDONE: BOOL;
	revs: REAL;
	valvePos: USINT;
	repli: INT:= 1;
	axiPower: MC_Power;
	i: INT;
	scale: FB_ScaleDevice;
	adjust: ARRAY[1..10] OF BOOL;
	correctRev: REAL;
	enableAdj: BOOL;
	opening: REAL;
	runLinear: BOOL;
	adjustSum: REAL;
	recResult: int:=1;
END_VAR

timeWt();
timer2();
timer3();

IF stop THEN
	powerOFF();
	stop:=FALSE;
END_IF

IF pumpNo = 1 OR pumpNo = 2 THEN
	valveNo:= 1;
ELSIF pumpNo = 3 OR pumpNo = 4 THEN
	valveNo:= 2;
ELSIF pumpNo = 5 OR pumpNo = 6 THEN
	valveNo:= 3;
ELSIF pumpNo = 7 OR pumpNo = 8 THEN
	valveNo:= 4;
ELSIF pumpNo = 9 OR pumpNo = 10 THEN
	valveNo:= 5;
END_IF

CASE state OF
	
0: //Idle
	IF start THEN
		GVL_Marco.revs:= GVL_Marco.mL_target;
		GVL_Marco.valvPos:= 6;
		timeWt(in:=TRUE, pt:=T#10S);
		repli:= 1;
		recResult:= 1;
		
		FOR i:= 1 TO 10 BY 1 DO
			GVL_Marco.resetAxi[i]:= FALSE;
			GVL_Marco.enableAxi[i]:= TRUE;
		END_FOR 
		
		FOR i:= 1 TO 5 BY 1 DO
			GVL_Marco.enableValv[i]:= TRUE;		
		END_FOR
		
		FOR i:=1 TO 50 BY 1 DO
			GVL_Marco.calibResult[i].grossWt:=0;
			GVL_Marco.calibResult[i].netWt:=0;
			GVL_Marco.calibResult[i].pumpNo:=0;
			GVL_Marco.calibResult[i].tareWt:=0;
		END_FOR
		
		state:= 10;
	ELSE
		state:= 0;
	END_IF
	
10:	//Enable the pump motor
	
	IF GVL_Motion.aValves[1].Axis.Status.InTargetPosition AND
		GVL_Motion.aValves[2].Axis.Status.InTargetPosition AND
		GVL_Motion.aValves[3].Axis.Status.InTargetPosition AND
		GVL_Motion.aValves[4].Axis.Status.InTargetPosition AND
		GVL_Motion.aValves[5].Axis.Status.InTargetPosition AND timeWt.Q THEN
		FOR i:= 1 TO 5 BY 1 DO
			GVL_Marco.enableValv[i]:= FALSE;		
		END_FOR
		timeWt(in:=FALSE);
		state:= 20;
	ELSE
		state:= 10;
	END_IF		

20:	//Fill the Jars from Box
	
	IF NOT GVL_Motion.aPumps[pumpNo].Rotary.Axis.Status.Disabled THEN
		
		revs:= GVL_Marco.revs*2;
		GVL_Marco.runFWD[pumpNo]:= TRUE;
		
		start:= FALSE;
		timer2(in:=TRUE, pt:=T#10S);
		state:= 30;
	ELSE
		state:= 20;
	END_IF

30: //Move valve to position 6
	
	IF NOT GVL_Motion.aPumps[pumpNo].Rotary.Axis.Status.Moving AND timer2.Q THEN
		
		GVL_Marco.valvPos:= 6;
		timer2(in:=FALSE);
		timeWt(in:=TRUE, pt:=T#10S);
		
		GVL_Marco.runFWD[pumpNo]:= FALSE;
		
		FOR i:=1 TO 5 BY 1 DO
			GVL_Marco.enableValv[i]:= TRUE;
		END_FOR
		
		
		state:= 40;
		
	ELSE
		state:= 30;
	END_IF


40: //Fill the calibration box(setup) - NO MORE

	IF GVL_Motion.aValves[1].Axis.Status.InTargetPosition AND
		GVL_Motion.aValves[2].Axis.Status.InTargetPosition AND
		GVL_Motion.aValves[3].Axis.Status.InTargetPosition AND
		GVL_Motion.aValves[4].Axis.Status.InTargetPosition AND
		GVL_Motion.aValves[5].Axis.Status.InTargetPosition AND timeWt.Q THEN
		
		FOR i:= 1 TO 5 BY 1 DO
			GVL_Marco.enableValv[i]:= FALSE;
		END_FOR
		
		//revs:= GVL_Marco.revs/2;
		//GVL_Marco.runBWD[pumpNo]:= TRUE;
		
		timeWt(in:=FALSE);
		timer2(in:=TRUE, pt:=T#10S);
		state:= 50;
		
	ELSE
		state:= 40;	
	END_IF

50: //Waiting

	IF NOT GVL_Motion.aPumps[pumpNo].Rotary.Axis.Status.Moving AND timer2.Q THEN
		GVL_Marco.runBWD[pumpNo]:= FALSE;
		timer2(in:=FALSE);
		timeWt(in:=TRUE, pt:=T#10S);
		GVL_Calibration.fbScaleDevice.RequestWeight();
		state:= 55;
	ELSE
		state:= 50;
	END_IF
	
55: //Make Tara
	
	IF timeWt.Q THEN
		tareWt:= GVL_Calibration.fbScaleDevice.RequestWeight();
		timeWt(in:=FALSE);
		state:= 60;
	ELSE
		state:= 55;
	END_IF
	
60: //Fill box from jar

	IF tareWt <> 9999.0 THEN
		GVL_Marco.calibResult[recResult].tareWt:= tareWt;
		revs:= GVL_Marco.revs;
		GVL_Marco.runBWD[pumpNo]:= TRUE;
		timer2(in:=TRUE, pt:=T#10S);
		state:= 70;
	ELSE
		state:= 60;
	END_IF
	
70: //Waiting

	IF NOT GVL_Motion.aPumps[pumpNo].Rotary.Axis.Status.Moving AND timer2.Q THEN
		GVL_Marco.runBWD[pumpNo]:= FALSE;
		timer2(in:=FALSE);
		timeWt(in:=TRUE, pt:=T#10S);
		GVL_Calibration.fbScaleDevice.RequestWeight();
		state:= 75;
	ELSE
		state:= 70;
	END_IF

75: //Get gross weight
	
	IF timeWt.Q THEN
		grossWt:= GVL_Calibration.fbScaleDevice.RequestWeight();
		timeWt(in:=FALSE);
		state:= 80;
	ELSE
		state:= 75;
	END_IF
	
80: //Return jar to box

	IF grossWt <> 9999.0 THEN
		GVL_Marco.calibResult[recResult].grossWt:= grossWt;
		GVL_Marco.calibResult[recResult].netWt:= GVL_Marco.calibResult[recResult].grossWt - GVL_Marco.calibResult[recResult].tareWt;
		GVL_Marco.calibResult[recResult].pumpNo:= pumpNo;
		recResult:= recResult +1;
			
		revs:= GVL_Marco.revs;
		GVL_Marco.runBWD[pumpNo]:= TRUE;

		timer3(in:=TRUE, pt:=T#10S);
		repli := repli +1; 
		state:= 90;
	ELSE
		state:= 80;
	END_IF

90: //Check replicates

	IF repli < replicates+1 AND timer3.Q AND GVL_Motion.aPumps[pumpNo].Rotary.Axis.Status.NotMoving THEN
		timer3(in:=FALSE);
		GVL_Marco.runBWD[pumpNo]:= FALSE;
		timer2(in:=TRUE, pt:=T#10S);
		state:= 50;
	ELSIF repli >= replicates AND timer3.Q AND GVL_Motion.aPumps[pumpNo].Rotary.Axis.Status.NotMoving THEN
		timer3(in:=FALSE);
		GVL_Marco.runBWD[pumpNo]:= FALSE;
		timer2(in:=TRUE, pt:=T#10S);
		state:= 100;
	ELSE
		state:= 90;
	END_IF

100: //Empty the jar to box

	IF  GVL_Motion.aValves[1].Axis.Status.InTargetPosition AND 
		GVL_Motion.aValves[2].Axis.Status.InTargetPosition AND
		GVL_Motion.aValves[3].Axis.Status.InTargetPosition AND
		GVL_Motion.aValves[4].Axis.Status.InTargetPosition AND
		GVL_Motion.aValves[5].Axis.Status.InTargetPosition AND timer2.Q THEN
		
		revs:= GVL_Marco.revs;
		IF pumpNo = 10 THEN
			GVL_Marco.runBWD[pumpNo]:= TRUE;
			state:= 110;
		ELSE
			pumpNo:= pumpNo + 1;
			repli:= 1;
			timer2(in:=TRUE, pt:=T#10S);
			state:= 20;
		END_IF
				
		timer2(in:=FALSE);
		timer3(in:=TRUE, pt:=T#10S);
		
	ELSE
		state:= 100;
	END_IF
	
110: //Done

	IF GVL_Motion.aPumps[1].Rotary.Axis.Status.NotMoving AND
		GVL_Motion.aPumps[2].Rotary.Axis.Status.NotMoving AND
		GVL_Motion.aPumps[3].Rotary.Axis.Status.NotMoving AND
		GVL_Motion.aPumps[4].Rotary.Axis.Status.NotMoving AND
		GVL_Motion.aPumps[5].Rotary.Axis.Status.NotMoving AND
		GVL_Motion.aPumps[6].Rotary.Axis.Status.NotMoving AND
		GVL_Motion.aPumps[7].Rotary.Axis.Status.NotMoving AND
		GVL_Motion.aPumps[8].Rotary.Axis.Status.NotMoving AND
		GVL_Motion.aPumps[9].Rotary.Axis.Status.NotMoving AND
		GVL_Motion.aPumps[10].Rotary.Axis.Status.NotMoving AND timer3.Q THEN
		FOR i:=1 TO 10 BY 1 DO
			GVL_Marco.runBWD[i]:= FALSE;
		END_FOR
		
		timer3(in:=FALSE);
		timeWt(in:=TRUE, pt:=T#10S);
		state:= 120;
	ELSE
		state:= 110;
	END_IF
	
120:

	IF GVL_Motion.aPumps[1].Rotary.Axis.Status.NotMoving AND
		GVL_Motion.aPumps[2].Rotary.Axis.Status.NotMoving AND
		GVL_Motion.aPumps[3].Rotary.Axis.Status.NotMoving AND
		GVL_Motion.aPumps[4].Rotary.Axis.Status.NotMoving AND
		GVL_Motion.aPumps[5].Rotary.Axis.Status.NotMoving AND
		GVL_Motion.aPumps[6].Rotary.Axis.Status.NotMoving AND
		GVL_Motion.aPumps[7].Rotary.Axis.Status.NotMoving AND
		GVL_Motion.aPumps[8].Rotary.Axis.Status.NotMoving AND
		GVL_Motion.aPumps[9].Rotary.Axis.Status.NotMoving AND
		GVL_Motion.aPumps[10].Rotary.Axis.Status.NotMoving AND timeWt.Q THEN
		FOR i:=1 TO 10 BY 1 DO
			GVL_Marco.resetAxi[i]:= TRUE;
			GVL_Marco.enableAxi[i]:= FALSE;
		END_FOR
		
		(*IF GVL_Marco.revs > GVL_Marco.mL_target THEN
			correctRev:= GVL_Marco.revs - GVL_Marco.mL_target;
		ELSIF GVL_Marco.revs < GVL_Marco.mL_target THEN
			correctRev:= GVL_Marco.mL_target - GVL_Marco.revs; 	
		END_IF*)
		state:= 0;
	ELSE
		state:= 120;
	END_IF
	
END_CASE

METHOD moveValve : BOOL
VAR
	state: INT;
	valveNo: INT;
END_VAR
VAR_INPUT
	pumNo: INT;
	valvePos: USINT;
	
END_VAR
IF pumpNo = 1 OR pumpNo = 2 THEN
	valveNo:= 1;
ELSIF pumpNo = 3 OR pumpNo = 4 THEN
	valveNo:= 2;
ELSIF pumpNo = 5 OR pumpNo = 6 THEN
	valveNo:= 3;
ELSIF pumpNo = 7 OR pumpNo = 8 THEN
	valveNo:= 4;
ELSIF pumpNo = 9 OR pumpNo = 10 THEN
	valveNo:= 5;
END_IF

GVL_Motion.aValvesObj[valveNo].MoveValve(iPosition := valvePos, rVelocity := GVL_Motion.aValves[1].rTargetVel, rAcc := GVL_Motion.aValves[1].rAcceleration, rDec := GVL_Motion.aValves[1].rDeceleration);

CASE state OF
	
0:

	IF NOT GVL_Motion.aValves[valveNo].Axis.Status.Moving THEN
		GVL_Motion.aValvesObj[valveNo].MoveValve(iPosition := valvePos, rVelocity := GVL_Motion.aValves[1].rTargetVel, rAcc := GVL_Motion.aValves[1].rAcceleration, rDec := GVL_Motion.aValves[1].rDeceleration);
		movimentDONE:=FALSE;
		state:= 1;
	ELSE
		state:= 0;	
	END_IF

1:
	IF NOT GVL_Motion.aValves[valveNo].Axis.Status.Moving THEN
			movimentDONE:= TRUE;
			State:= 0;
		ELSE
			state:= 1;
		END_IF
	
	
END_CASE
END_METHOD

METHOD powerOFF : BOOL
VAR
	axiPower: MC_Power;
	pumpNo: INT;
	
END_VAR
VAR_INPUT
	
	
END_VAR
FOR pumpNo:=1 TO 10 BY 1 DO
	axiPower(
	Axis:= GVL_Motion.aPumps[pumpNo].Rotary.Axis,
	Enable:= FALSE,
	Enable_Negative:= FALSE,
	Enable_Positive:= FALSE,
	Override:= 100);
	
	axiPower(
	Axis:= GVL_Motion.aPumps[pumpNo].Linear.Axis,
	Enable:= FALSE,
	Enable_Negative:= FALSE,
	Enable_Positive:= FALSE,
	Override:= 100);
END_FOR
END_METHOD

METHOD runBwd : BOOL
VAR
	moveRel: MC_MoveRelative;
	selectPosRel: LREAL;
	
END_VAR
VAR_INPUT
	pumpNo: INT;
	revs: INT;
	 
END_VAR

selectPosRel:= revs*360;

moveRel(
	Axis:= GVL_Motion.aPumps[pumpNo].Rotary.Axis,
	Execute:= TRUE,
	Distance:= selectPosRel*-1,
	Velocity:= 3000,
	Acceleration:= 3000,
	Deceleration:= 3000);
END_METHOD

METHOD runFwd : BOOL
VAR
	moveRel: MC_MoveRelative;
	selectPosRel: LREAL;
	
END_VAR
VAR_INPUT
	pumpNo: INT;
	revs: INT;
	 
END_VAR

selectPosRel:= revs*360;

moveRel(
	Axis:= GVL_Motion.aPumps[pumpNo].Rotary.Axis,
	Execute:= TRUE,
	Distance:= selectPosRel,
	Velocity:= 3000,
	Acceleration:= 3000,
	Deceleration:= 3000);
END_METHOD

END_PROGRAM

// ---- VISUs/GlobalTextList.TcGTLO
TEXTLIST GlobalTextList
  18 = 'dddddd'
  748 = 'Error Ack'
  1 = 'Reset BT'
END_TEXTLIST

// ---- VISUs/Visualization.TcVIS
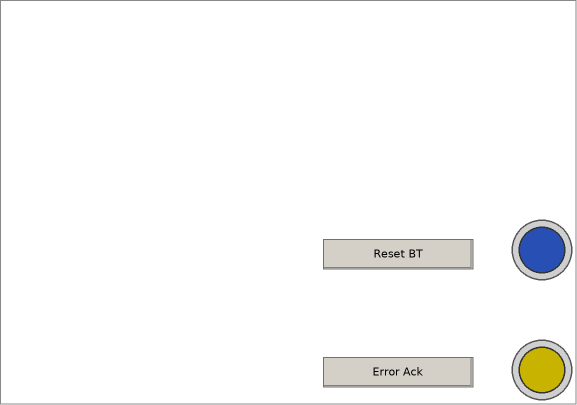
VISUALIZATION Visualization  // 577x405
    Button (323,239 150x30), "Reset BT", pressed state: GVL_Safety.bResetButtonVISU
        OnMouseClick: toggle GVL_Safety.bResetButtonVISU
    Lamp1 (507,215 70x70), variable: GVL_Safety.bResetButtonVISU, style: Lamp-Lamp1-Blue
    Button (323,357 150x30), "Error Ack", pressed state: GVL_Safety.bAckButtonVISU
        OnMouseClick: toggle GVL_Safety.bAckButtonVISU
    Lamp1 (507,335 70x70), variable: GVL_Safety.bSafetyErrorAck, style: Lamp-Lamp1-Yellow
END_VISUALIZATION
